// TIA Portal project "COMPACTADOR" (V21)

(* hardware
DEVICE "S7-1200 station_1"  S7-1200 Station
   slot 0: "Rack_0"  S7-1200 Rack  Rack  V1.0
   slot 1: "PLC_1"  CPU 1214C DC/DC/DC  6ES7 214-1AG40-0XB0  V4.6
   slot 2: "DI 16x24VDC_1"  SM 1221 DI16 x 24VDC  6ES7 221-1BH32-0XB0  V2.0
   slot 3: "DI 16x24VDC_2"  SM 1221 DI16 x 24VDC  6ES7 221-1BH32-0XB0  V2.0
   slot 4: "DI 16x24VDC_3"  SM 1221 DI16 x 24VDC  6ES7 221-1BH32-0XB0  V2.0
   slot 5: "DQ 16xRelay_1"  SM 1222 DQ16 x relay  6ES7 222-1HH32-0XB0  V2.0
*)

// ===== PLC "PLC_1"  CPU 1214C DC/DC/DC =====

VAR_GLOBAL   // PLC tag table "Default tag table"
   "Name" AT Logical Address : Data Type;   // Comment
END_VAR

VAR_GLOBAL   // PLC tag table "Entradas_CPU_Local"
   "STOP7" AT %I0.0 : Bool;   // Paragem Local / Botao Cogumelo de Paragem Geral (Contacto NF)
   "START" AT %I0.1 : Bool;   // Botao de Arranque do Sistema (Contacto NA)
   "AVANCA" AT %I0.2 : Bool;   // Botao Manual de Avanco do Cilindro Hidraulico (Contacto NA)
   "RECUA" AT %I0.3 : Bool;   // Botao Manual de Recuo do Cilindro Hidraulico (Contacto NA)
   "FR1" AT %I0.4 : Bool;   // Disparo / Auxiliar do Rele Termico do Motor M1 (Contacto NF)
   "FR2" AT %I0.5 : Bool;   // Disparo / Auxiliar do Rele Termico do Motor M2 (Contacto NF)
   "FR3" AT %I0.6 : Bool;   // Disparo / Auxiliar do Rele Termico do Motor M3 (Contacto NF)
   "FR4" AT %I0.7 : Bool;   // Disparo / Auxiliar do Rele Termico do Motor M4 (Contacto NF)
   "FR5" AT %I1.0 : Bool;   // Disparo / Auxiliar do Rele Termico do Motor M5 (Contacto NF)
   "FR6" AT %I1.1 : Bool;   // Disparo / Auxiliar do Rele Termico da Bomba M6 (Contacto NF)
   "SEL_AUTO" AT %I1.2 : Bool;   // Chave Seletora Auto/Manual - Posicao Automatico (Contacto NA)
   "SEL_MANUAL" AT %I1.3 : Bool;   // Chave Seletora Auto/Manual - Posicao Manual (Contacto NA)
   "RESERVA_I1_4" AT %I1.4 : Bool;   // Reserva Tecnica Local CPU
   "RESERVA_I1_5" AT %I1.5 : Bool;   // Reserva Tecnica Local CPU
END_VAR

VAR_GLOBAL   // PLC tag table "Entradas_Expansao1_SM1221"
   "SIN_Y7_COMP" AT %I2.0 : Bool;   // Diagnostico de Seguranca do Compactador (Rele IFM Y7)
   "NA_S1_COMP" AT %I2.1 : Bool;   // Interlock / Fim de Curso de Seguranca 1 do Compactador
   "NA_S2_COMP" AT %I2.2 : Bool;   // Interlock / Fim de Curso de Seguranca 2 do Compactador
   "NA_S3_COMP" AT %I2.3 : Bool;   // Interlock / Fim de Curso de Seguranca 3 do Compactador
   "SIN_Y7_M1" AT %I2.4 : Bool;   // Diagnostico de Seguranca do Motor M1 (Rele IFM Y7)
   "NA_STOP_M1" AT %I2.5 : Bool;   // Botao / Paragem Local de Seguranca do Tapete M1
   "SIN_Y7_M2" AT %I2.6 : Bool;   // Diagnostico de Seguranca do Motor M2 (Rele IFM Y7)
   "SIN_Y7_M3" AT %I2.7 : Bool;   // Diagnostico de Seguranca do Motor M3 (Rele IFM Y7)
   "NA_STOP_M2" AT %I3.0 : Bool;   // Botao / Paragem Local de Seguranca do Tapete M2
   "NA_STOP_M3" AT %I3.1 : Bool;   // Botao / Paragem Local de Seguranca do Tapete M3
   "SIN_Y7_M4" AT %I3.2 : Bool;   // Diagnostico de Seguranca do Motor M4 (Rele IFM Y7)
   "NA_STOP_M4" AT %I3.3 : Bool;   // Botao / Paragem Local de Seguranca do Tapete M4
   "SIN_Y7_M5" AT %I3.4 : Bool;   // Diagnostico de Seguranca do Motor M5 (Rele IFM Y7)
   "NA_STOP_M5" AT %I3.5 : Bool;   // Botao / Paragem Local de Seguranca do Tapete M5
   "SENSOR_75_PERCENT" AT %I3.6 : Bool;   // Sensor Optoeletronico de Nivel da Moega a 75%
   "SENSOR_100_PERCENT" AT %I3.7 : Bool;   // Sensor Optoeletronico de Nivel da Moega a 100%
END_VAR

VAR_GLOBAL   // PLC tag table "Entradas_Expansao2_SM1221"
   "M1_S4" AT %I4.0 : Bool;   // Grupo Motor M1 (Tapete 1) - Sensor S4 de Posicao / Presenca
   "M1_S5" AT %I4.1 : Bool;   // Grupo Motor M1 (Tapete 1) - Sensor S5 de Posicao / Presenca
   "M1_S6" AT %I4.2 : Bool;   // Grupo Motor M1 (Tapete 1) - Sensor S6 de Posicao / Presenca
   "M2_S7" AT %I4.3 : Bool;   // Grupo Motor M2 (Tapete 2) - Sensor S7 de Posicao / Presenca
   "M2_S8" AT %I4.4 : Bool;   // Grupo Motor M2 (Tapete 2) - Sensor S8 de Posicao / Presenca
   "M2_S9" AT %I4.5 : Bool;   // Grupo Motor M2 (Tapete 2) - Sensor S9 de Posicao / Presenca
   "M3_S10" AT %I4.6 : Bool;   // Grupo Motor M3 (Tapete 3) - Sensor S10 de Posicao / Presenca
   "M3_S11" AT %I4.7 : Bool;   // Grupo Motor M3 (Tapete 3) - Sensor S11 de Posicao / Presenca
   "M3_S12" AT %I5.0 : Bool;   // Grupo Motor M3 (Tapete 3) - Sensor S12 de Posicao / Presenca
   "M4_S13" AT %I5.1 : Bool;   // Grupo Motor M4 (Tapete 4) - Sensor S13 de Posicao / Presenca
   "M4_S14" AT %I5.2 : Bool;   // Grupo Motor M4 (Tapete 4) - Sensor S14 de Posicao / Presenca
   "M4_S15" AT %I5.3 : Bool;   // Grupo Motor M4 (Tapete 4) - Sensor S15 de Posicao / Presenca
   "M5_S16" AT %I5.4 : Bool;   // Grupo Motor M5 (Tapete 5) - Sensor S16 de Posicao / Presenca
   "M5_S17" AT %I5.5 : Bool;   // Grupo Motor M5 (Tapete 5) - Sensor S17 de Posicao / Presenca
   "M5_S18" AT %I5.6 : Bool;   // Grupo Motor M5 (Tapete 5) - Sensor S18 de Posicao / Presenca
   "M5_S19" AT %I5.7 : Bool;   // Grupo Motor M5 (Tapete 5) - Sensor S19 de Posicao / Presenca
END_VAR

VAR_GLOBAL   // PLC tag table "Entradas_Expansao3_SM1221"
   "S20_COMP" AT %I6.0 : Bool;   // Sensor de Proximidade Adicional 20 do Compactador
   "S21_COMP" AT %I6.1 : Bool;   // Sensor de Proximidade Adicional 21 do Compactador
   "STOP6_GERAL" AT %I6.2 : Bool;   // Paragem Local / Botao Cogumelo de Paragem Geral (Contacto NF)
   "RESERVA_I6_5" AT %I6.5 : Bool;   // Reserva Tecnica Modulo DI 3
   "RESERVA_I6_6" AT %I6.6 : Bool;   // Reserva Tecnica Modulo DI 3
   "RESERVA_I6_7" AT %I6.7 : Bool;   // Reserva Tecnica Modulo DI 3
   "RESERVA_I7_0" AT %I7.0 : Bool;   // Reserva Tecnica Modulo DI 3
   "RESERVA_I7_1" AT %I7.1 : Bool;   // Reserva Tecnica Modulo DI 3
   "RESERVA_I7_2" AT %I7.2 : Bool;   // Reserva Tecnica Modulo DI 3
   "RESERVA_I7_3" AT %I7.3 : Bool;   // Reserva Tecnica Modulo DI 3
   "RESERVA_I7_4" AT %I7.4 : Bool;   // Reserva Tecnica Modulo DI 3
   "RESERVA_I7_5" AT %I7.5 : Bool;   // Reserva Tecnica Modulo DI 3
   "RESERVA_I7_6" AT %I7.6 : Bool;   // Reserva Tecnica Modulo DI 3
   "RESERVA_I7_7" AT %I7.7 : Bool;   // Reserva Tecnica Modulo DI 3
   "NA_STOP_COMP" AT %I6.3 : Bool;   // Botao / Paragem Local de Seguranca do Compactador
   "RESERVA_I6_4" AT %I6.4 : Bool;   // Reserva Tecnica Modulo DI 3
END_VAR

VAR_GLOBAL   // PLC tag table "Saidas_CPU_Local"
   "KM1" AT %Q0.0 : Bool;   // Contactor de Processo do Motor M1 (Tapete 1)
   "KM2" AT %Q0.1 : Bool;   // Contactor de Processo do Motor M2 (Tapete 2)
   "KM3" AT %Q0.2 : Bool;   // Contactor de Processo do Motor M3 (Tapete 3)
   "KM4" AT %Q0.3 : Bool;   // Contactor de Processo do Motor M4 (Tapete 4)
   "KM5" AT %Q0.4 : Bool;   // Contactor de Processo do Motor M5 (Tapete 5)
   "START_SS_M6" AT %Q0.5 : Bool;   // Sinal de Habilitacao / Start da Soft Starter (Bomba M6)
   "Y1_AVANCA" AT %Q0.6 : Bool;   // Eletrovalvula de Avanco do Cilindro Hidraulico
   "Y2_RECUA" AT %Q0.7 : Bool;   // Eletrovalvula de Recuo do Cilindro Hidraulico
   "H1_VERDE" AT %Q1.0 : Bool;   // Sinalizador Luminoso Verde: Linha em Funcionamento / Automatico
   "H2_AMARELO" AT %Q1.1 : Bool;   // Sinalizador Luminoso Amarelo: Estado de Prontidao / Standby
END_VAR

VAR_GLOBAL   // PLC tag table "Saidas_Expansao1_SM1222"
   "H13_AUTO" AT %Q2.0 : Bool;   // Sinalizador: Modo AUTOMATICO Selecionado
   "H14_MANUAL" AT %Q2.1 : Bool;   // Sinalizador: Modo MANUAL Selecionado
   "H3_AZUL" AT %Q2.3 : Bool;   // Sinalizador Azul: Nivel da Moega a 75%
   "H4_VERMELHO" AT %Q2.4 : Bool;   // Sinalizador Vermelho: Nivel da Moega a 100%
   "H5_VERMELHO" AT %Q2.5 : Bool;   // Sinalizador Vermelho: Paragem / Avaria Geral da Linha
   "H6_VERMELHO" AT %Q2.6 : Bool;   // Sinalizador Vermelho: Paragem / Avaria do Compactador
   "H7_VERMELHO" AT %Q2.7 : Bool;   // Sinalizador Vermelho: Paragem / Avaria do Motor M1
   "H8_VERMELHO" AT %Q3.0 : Bool;   // Sinalizador Vermelho: Paragem / Avaria do Motor M2
   "H9_VERMELHO" AT %Q3.1 : Bool;   // Sinalizador Vermelho: Paragem / Avaria do Motor M3
   "H10_VERMELHO" AT %Q3.2 : Bool;   // Sinalizador Vermelho: Paragem / Avaria do Motor M4
   "H11_VERMELHO" AT %Q3.3 : Bool;   // Sinalizador Vermelho: Paragem / Avaria do Motor M5
   "H12_VERMELHO" AT %Q3.4 : Bool;   // Sinalizador Vermelho: Paragem / Avaria da Bomba M6
   "RESERVA_Q2_2" AT %Q2.2 : Bool;   // Reserva Tecnica Modulo DQ 1
   "RESERVA_Q3_5" AT %Q3.5 : Bool;   // Reserva Tecnica Modulo DQ 1
   "RESERVA_Q3_6" AT %Q3.6 : Bool;   // Reserva Tecnica Modulo DQ 1
   "RESERVA_Q3_7" AT %Q3.7 : Bool;   // Reserva Tecnica Modulo DQ 1
END_VAR

VAR_GLOBAL   // PLC tag table "Marcadores_Internos"
   "OK_SISTEMA" AT %M0.0 : Bool;   // Permissivo geral do sistema (calculado em FC1)
   "AUT_LINHA_LIGADA" AT %M0.1 : Bool;   // Selo da linha em modo automatico (FC3)
   "MODO_MANUAL" AT %M0.2 : Bool;   // Modo manual selecionado (FC2)
   "CICLO_RECUO" AT %M0.3 : Bool;   // Ciclo de recuo do cilindro hidraulico (FC4)
   "EMERGENCIA" AT %M0.4 : Bool;   // Paragem de emergencia ativa (FC1)
   "ETAPA_GRAFCET" AT %MW2 : Word;   // Variavel de etapa atual do GRAFCET (FC5_GRAFCET)
   "INATIVIDADE_ATIVA" AT %M0.5 : Bool;   // Timer de inatividade ativo; linha sem material durante 30 s
END_VAR

DATA_BLOCK "DB_LinhaCompactador"   // DB1
{ S7_Optimized_Access := 'TRUE' }
VERSION : 0.1
// stored: InstanceOfName FB_LinhaCompactador
"FB_LinhaCompactador"
BEGIN
END_DATA_BLOCK

FUNCTION_BLOCK "FB_LinhaCompactador"   // FB1, SCL
{ S7_Optimized_Access := 'TRUE' }
VERSION : 0.1
   VAR
      T_Start_M6 : TON_TIME;
      T_Start_M5 : TON_TIME;
      T_Start_M34 : TON_TIME;
      T_Stop_M12 : TON_TIME;
      T_Stop_M34 : TON_TIME;
      T_Stop_M5 : TON_TIME;
      T_Inatividade : TON_TIME;
   END_VAR
   VAR_TEMP
      AutoOk : Bool;
      FaultM1 : Bool;
      FaultM2 : Bool;
      FaultM3 : Bool;
      FaultM4 : Bool;
      FaultM5 : Bool;
      FaultM6 : Bool;
      FaultComp : Bool;
      EmptyM3M4 : Bool;
      EmptyM5 : Bool;
      ManualMove : Bool;
      FrontFreeM1 : Bool;
      FrontFreeM2 : Bool;
      FrontFreeM3 : Bool;
      FrontFreeM4 : Bool;
      FrontFreeM5 : Bool;
      ContentorLivre : Bool;
      LinhaSemMaterial : Bool;
   END_VAR
BEGIN

       // FC1 - Seguranca geral
       "OK_SISTEMA" :=
           "STOP7" AND
           "STOP6_GERAL" AND
           "FR1" AND
           "FR2" AND
           "FR3" AND
           "FR4" AND
           "FR5" AND
           "FR6" AND
           "SIN_Y7_COMP" AND
           "SIN_Y7_M1" AND
           "SIN_Y7_M2" AND
           "SIN_Y7_M3" AND
           "SIN_Y7_M4" AND
           "SIN_Y7_M5" AND
           "NA_STOP_M1" AND
           "NA_STOP_M2" AND
           "NA_STOP_M3" AND
           "NA_STOP_M4" AND
           "NA_STOP_M5" AND
           "NA_STOP_COMP";

       "EMERGENCIA" := NOT "OK_SISTEMA";

       // FC2 - Selecao de modo
       #AutoOk := "SEL_AUTO" AND NOT "SEL_MANUAL" AND "OK_SISTEMA";
       "MODO_MANUAL" := "SEL_MANUAL" AND NOT "SEL_AUTO" AND "OK_SISTEMA";
       "H13_AUTO" := "SEL_AUTO" AND NOT "SEL_MANUAL";
       "H14_MANUAL" := "SEL_MANUAL" AND NOT "SEL_AUTO";

       // Diagnosticos por grupo
       #FaultM1 := NOT "FR1" OR NOT "NA_STOP_M1" OR NOT "SIN_Y7_M1";
       #FaultM2 := NOT "FR2" OR NOT "NA_STOP_M2" OR NOT "SIN_Y7_M2";
       #FaultM3 := NOT "FR3" OR NOT "NA_STOP_M3" OR NOT "SIN_Y7_M3";
       #FaultM4 := NOT "FR4" OR NOT "NA_STOP_M4" OR NOT "SIN_Y7_M4";
       #FaultM5 := NOT "FR5" OR NOT "NA_STOP_M5" OR NOT "SIN_Y7_M5";
       #FaultM6 := NOT "FR6";
       #FaultComp := NOT "NA_STOP_COMP" OR NOT "SIN_Y7_COMP";

       // FC6 - Nivel da moega
       "H3_AZUL" := "SENSOR_75_PERCENT";
       "H4_VERMELHO" := "SENSOR_100_PERCENT";

       #EmptyM3M4 :=
           NOT "M3_S10" AND NOT "M3_S11" AND NOT "M3_S12" AND
           NOT "M4_S13" AND NOT "M4_S14" AND NOT "M4_S15";

       #EmptyM5 :=
           NOT "M5_S16" AND NOT "M5_S17" AND NOT "M5_S18" AND NOT "M5_S19";

       #ManualMove := "MODO_MANUAL" AND (("AVANCA" AND NOT "RECUA") OR ("RECUA" AND NOT "AVANCA"));

       // Anti-acumulacao / anti-queda: o tapete de tras so alimenta se a zona da frente estiver livre.
       #FrontFreeM1 := NOT "M3_S10" AND NOT "M3_S11" AND NOT "M3_S12";
       #FrontFreeM2 := NOT "M4_S13" AND NOT "M4_S14" AND NOT "M4_S15";
       #FrontFreeM3 := NOT "M5_S16" AND NOT "M5_S17";
       #FrontFreeM4 := NOT "M5_S18" AND NOT "M5_S19";
       #FrontFreeM5 := NOT "SENSOR_100_PERCENT";
       #ContentorLivre := NOT "S20_COMP" AND NOT "S21_COMP";
       #LinhaSemMaterial :=
           NOT "M1_S4" AND NOT "M1_S5" AND NOT "M1_S6" AND
           NOT "M2_S7" AND NOT "M2_S8" AND NOT "M2_S9" AND
           NOT "M3_S10" AND NOT "M3_S11" AND NOT "M3_S12" AND
           NOT "M4_S13" AND NOT "M4_S14" AND NOT "M4_S15" AND
           NOT "M5_S16" AND NOT "M5_S17" AND NOT "M5_S18" AND NOT "M5_S19" AND
           NOT "S20_COMP" AND NOT "S21_COMP" AND
           NOT "SENSOR_75_PERCENT" AND NOT "SENSOR_100_PERCENT";

       // Timers de arranque/paragem em cascata
       #T_Start_M6(IN := (#AutoOk AND #ContentorLivre AND ("ETAPA_GRAFCET" = WORD#16#000A)), PT := T#3s);
       #T_Start_M5(IN := (#AutoOk AND #ContentorLivre AND ("ETAPA_GRAFCET" = WORD#16#0014)), PT := T#2s);
       #T_Start_M34(IN := (#AutoOk AND #ContentorLivre AND ("ETAPA_GRAFCET" = WORD#16#001E)), PT := T#2s);
       #T_Stop_M12(IN := ("ETAPA_GRAFCET" = WORD#16#0064), PT := T#2s);
       #T_Stop_M34(IN := ("ETAPA_GRAFCET" = WORD#16#006E), PT := T#2s);
       #T_Stop_M5(IN := ("ETAPA_GRAFCET" = WORD#16#0078), PT := T#2s);
       #T_Inatividade(IN := (#AutoOk AND "AUT_LINHA_LIGADA" AND #LinhaSemMaterial), PT := T#30s);
       "INATIVIDADE_ATIVA" := #T_Inatividade.Q;

       // Prioridade maxima: emergencia ou modo invalido
       IF "EMERGENCIA" OR ("SEL_AUTO" AND "SEL_MANUAL") THEN
           "KM1" := FALSE;
           "KM2" := FALSE;
           "KM3" := FALSE;
           "KM4" := FALSE;
           "KM5" := FALSE;
           "START_SS_M6" := FALSE;
           "Y1_AVANCA" := FALSE;
           "Y2_RECUA" := FALSE;
           "AUT_LINHA_LIGADA" := FALSE;
           "CICLO_RECUO" := FALSE;
           "ETAPA_GRAFCET" := WORD#16#0000;

       ELSIF "MODO_MANUAL" THEN
           // FC4 - Manual do compactador, com intertravamento avanca/recuo
           "AUT_LINHA_LIGADA" := FALSE;
           "ETAPA_GRAFCET" := WORD#16#0000;
           "KM1" := FALSE;
           "KM2" := FALSE;
           "KM3" := FALSE;
           "KM4" := FALSE;
           "KM5" := FALSE;
           "START_SS_M6" := #ManualMove;
           "Y1_AVANCA" := "AVANCA" AND NOT "RECUA" AND "OK_SISTEMA";
           "Y2_RECUA" := "RECUA" AND NOT "AVANCA" AND "OK_SISTEMA";

       ELSIF #AutoOk THEN
           // FC3 - Automatico com arranque/paragem em cascata
           IF ("ETAPA_GRAFCET" = WORD#16#0000) AND "START" AND NOT "SENSOR_100_PERCENT" AND #ContentorLivre THEN
               "ETAPA_GRAFCET" := WORD#16#000A;
           END_IF;

           IF (("ETAPA_GRAFCET" = WORD#16#0028) AND (NOT "SEL_AUTO" OR "SENSOR_100_PERCENT" OR "INATIVIDADE_ATIVA")) THEN
               "ETAPA_GRAFCET" := WORD#16#0064;
           END_IF;

           IF ("ETAPA_GRAFCET" = WORD#16#000A) AND #T_Start_M6.Q THEN
               "ETAPA_GRAFCET" := WORD#16#0014;
           ELSIF ("ETAPA_GRAFCET" = WORD#16#0014) AND #T_Start_M5.Q THEN
               "ETAPA_GRAFCET" := WORD#16#001E;
           ELSIF ("ETAPA_GRAFCET" = WORD#16#001E) AND #T_Start_M34.Q THEN
               "ETAPA_GRAFCET" := WORD#16#0028;
               "AUT_LINHA_LIGADA" := TRUE;
           ELSIF ("ETAPA_GRAFCET" = WORD#16#0064) AND (#T_Stop_M12.Q OR #EmptyM3M4) THEN
               "ETAPA_GRAFCET" := WORD#16#006E;
           ELSIF ("ETAPA_GRAFCET" = WORD#16#006E) AND (#T_Stop_M34.Q OR #EmptyM5) THEN
               "ETAPA_GRAFCET" := WORD#16#0078;
           ELSIF ("ETAPA_GRAFCET" = WORD#16#0078) AND #T_Stop_M5.Q THEN
               "ETAPA_GRAFCET" := WORD#16#0000;
               "AUT_LINHA_LIGADA" := FALSE;
           END_IF;

           "START_SS_M6" := ("ETAPA_GRAFCET" <> WORD#16#0000) AND NOT #FaultM6 AND NOT #FaultComp;

           "KM5" :=
               (("ETAPA_GRAFCET" = WORD#16#0014) OR
                ("ETAPA_GRAFCET" = WORD#16#001E) OR
                ("ETAPA_GRAFCET" = WORD#16#0028) OR
                ("ETAPA_GRAFCET" = WORD#16#0064) OR
                ("ETAPA_GRAFCET" = WORD#16#006E)) AND
               #ContentorLivre AND
               #FrontFreeM5 AND
               NOT #FaultM5;

           "KM3" :=
               (("ETAPA_GRAFCET" = WORD#16#001E) OR
                ("ETAPA_GRAFCET" = WORD#16#0028) OR
                ("ETAPA_GRAFCET" = WORD#16#0064)) AND
               #ContentorLivre AND
               #FrontFreeM3 AND
               NOT #FaultM3 AND NOT #FaultM5;

           "KM4" :=
               (("ETAPA_GRAFCET" = WORD#16#001E) OR
                ("ETAPA_GRAFCET" = WORD#16#0028) OR
                ("ETAPA_GRAFCET" = WORD#16#0064)) AND
               #ContentorLivre AND
               #FrontFreeM4 AND
               NOT #FaultM4 AND NOT #FaultM5;

           "KM1" :=
               ("ETAPA_GRAFCET" = WORD#16#0028) AND
               #ContentorLivre AND
               NOT "SENSOR_100_PERCENT" AND
               #FrontFreeM1 AND
               NOT #FaultM1 AND NOT #FaultM3 AND NOT #FaultM5;

           "KM2" :=
               ("ETAPA_GRAFCET" = WORD#16#0028) AND
               #ContentorLivre AND
               NOT "SENSOR_100_PERCENT" AND
               #FrontFreeM2 AND
               NOT #FaultM2 AND NOT #FaultM4 AND NOT #FaultM5;

           // Ciclo basico do compactador. S20/S21 monitoram o contentor e nao sao fins de curso.
           IF "NA_S2_COMP" THEN
               "CICLO_RECUO" := TRUE;
           ELSIF "NA_S1_COMP" THEN
               "CICLO_RECUO" := FALSE;
           END_IF;

           "Y1_AVANCA" := "START_SS_M6" AND NOT "CICLO_RECUO" AND NOT "NA_S2_COMP";
           "Y2_RECUA" := "START_SS_M6" AND "CICLO_RECUO" AND NOT "NA_S1_COMP";

       ELSE
           // Sem modo valido: saidas desligadas, sistema em standby.
           "KM1" := FALSE;
           "KM2" := FALSE;
           "KM3" := FALSE;
           "KM4" := FALSE;
           "KM5" := FALSE;
           "START_SS_M6" := FALSE;
           "Y1_AVANCA" := FALSE;
           "Y2_RECUA" := FALSE;
           "AUT_LINHA_LIGADA" := FALSE;
           "ETAPA_GRAFCET" := WORD#16#0000;
       END_IF;

       // FC7 - Sinalizacao
       "H1_VERDE" := #AutoOk AND "AUT_LINHA_LIGADA" AND #ContentorLivre;
       "H2_AMARELO" := "OK_SISTEMA" AND (NOT "AUT_LINHA_LIGADA" OR NOT #ContentorLivre);
       "H6_VERMELHO" := #FaultComp;
       "H7_VERMELHO" := #FaultM1;
       "H8_VERMELHO" := #FaultM2;
       "H9_VERMELHO" := #FaultM3;
       "H10_VERMELHO" := #FaultM4;
       "H11_VERMELHO" := #FaultM5;
       "H12_VERMELHO" := #FaultM6;
       "H5_VERMELHO" :=
           "EMERGENCIA" OR
           ("SEL_AUTO" AND "SEL_MANUAL") OR
           #FaultComp OR #FaultM1 OR #FaultM2 OR #FaultM3 OR #FaultM4 OR #FaultM5 OR #FaultM6;
END_FUNCTION_BLOCK

FUNCTION "FC_LinhaCompactador_LAD" : Void   // FC21, LAD
{ S7_Optimized_Access := 'TRUE' }
VERSION : 0.1
// Visualizacao LAD da logica principal. A sequencia temporizada executavel continua em FB_LinhaCompactador.
BEGIN

REGION Network 1: FC1 - OK_SISTEMA: cadeia geral de seguranca
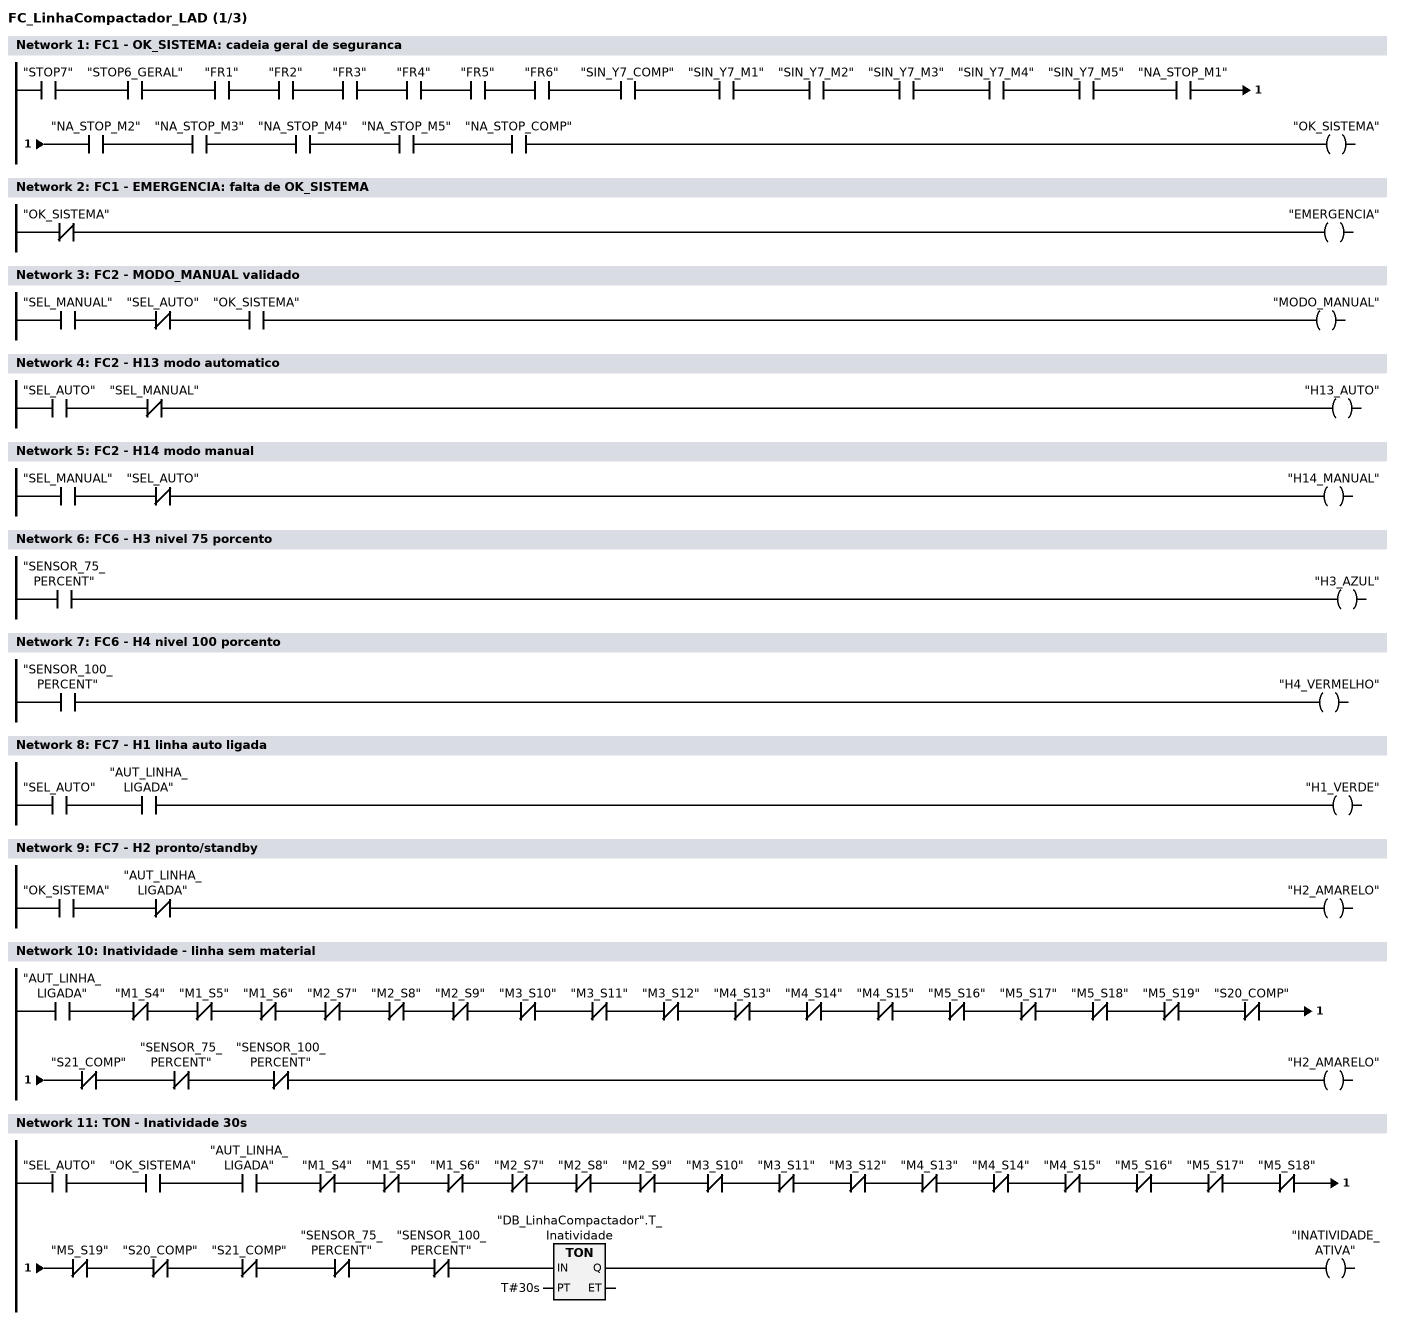
   RUNG wire#powerrail
      Contact( "STOP7" )
      Contact( "STOP6_GERAL" )
      Contact( "FR1" )
      Contact( "FR2" )
      Contact( "FR3" )
      Contact( "FR4" )
      Contact( "FR5" )
      Contact( "FR6" )
      Contact( "SIN_Y7_COMP" )
      Contact( "SIN_Y7_M1" )
      Contact( "SIN_Y7_M2" )
      Contact( "SIN_Y7_M3" )
      Contact( "SIN_Y7_M4" )
      Contact( "SIN_Y7_M5" )
      Contact( "NA_STOP_M1" )
      Contact( "NA_STOP_M2" )
      Contact( "NA_STOP_M3" )
      Contact( "NA_STOP_M4" )
      Contact( "NA_STOP_M5" )
      Contact( "NA_STOP_COMP" )
      Coil( "OK_SISTEMA" )
   END_RUNG
   // the same network as SCL:
   "OK_SISTEMA" := "STOP7" AND "STOP6_GERAL" AND "FR1" AND "FR2" AND "FR3" AND "FR4" AND "FR5" AND "FR6" AND "SIN_Y7_COMP" AND "SIN_Y7_M1" AND "SIN_Y7_M2" AND "SIN_Y7_M3" AND "SIN_Y7_M4" AND "SIN_Y7_M5" AND "NA_STOP_M1" AND "NA_STOP_M2" AND "NA_STOP_M3" AND "NA_STOP_M4" AND "NA_STOP_M5" AND "NA_STOP_COMP";
END_REGION

REGION Network 2: FC1 - EMERGENCIA: falta de OK_SISTEMA
   RUNG wire#powerrail
      I_Contact( "OK_SISTEMA" )
      Coil( "EMERGENCIA" )
   END_RUNG
   // the same network as SCL:
   "EMERGENCIA" := NOT "OK_SISTEMA";
END_REGION

REGION Network 3: FC2 - MODO_MANUAL validado
   RUNG wire#powerrail
      Contact( "SEL_MANUAL" )
      I_Contact( "SEL_AUTO" )
      Contact( "OK_SISTEMA" )
      Coil( "MODO_MANUAL" )
   END_RUNG
   // the same network as SCL:
   "MODO_MANUAL" := "SEL_MANUAL" AND NOT "SEL_AUTO" AND "OK_SISTEMA";
END_REGION

REGION Network 4: FC2 - H13 modo automatico
   RUNG wire#powerrail
      Contact( "SEL_AUTO" )
      I_Contact( "SEL_MANUAL" )
      Coil( "H13_AUTO" )
   END_RUNG
   // the same network as SCL:
   "H13_AUTO" := "SEL_AUTO" AND NOT "SEL_MANUAL";
END_REGION

REGION Network 5: FC2 - H14 modo manual
   RUNG wire#powerrail
      Contact( "SEL_MANUAL" )
      I_Contact( "SEL_AUTO" )
      Coil( "H14_MANUAL" )
   END_RUNG
   // the same network as SCL:
   "H14_MANUAL" := "SEL_MANUAL" AND NOT "SEL_AUTO";
END_REGION

REGION Network 6: FC6 - H3 nivel 75 porcento
   RUNG wire#powerrail
      Contact( "SENSOR_75_PERCENT" )
      Coil( "H3_AZUL" )
   END_RUNG
   // the same network as SCL:
   "H3_AZUL" := "SENSOR_75_PERCENT";
END_REGION

REGION Network 7: FC6 - H4 nivel 100 porcento
   RUNG wire#powerrail
      Contact( "SENSOR_100_PERCENT" )
      Coil( "H4_VERMELHO" )
   END_RUNG
   // the same network as SCL:
   "H4_VERMELHO" := "SENSOR_100_PERCENT";
END_REGION

REGION Network 8: FC7 - H1 linha auto ligada
   RUNG wire#powerrail
      Contact( "SEL_AUTO" )
      Contact( "AUT_LINHA_LIGADA" )
      Coil( "H1_VERDE" )
   END_RUNG
   // the same network as SCL:
   "H1_VERDE" := "SEL_AUTO" AND "AUT_LINHA_LIGADA";
END_REGION

REGION Network 9: FC7 - H2 pronto/standby
   RUNG wire#powerrail
      Contact( "OK_SISTEMA" )
      I_Contact( "AUT_LINHA_LIGADA" )
      Coil( "H2_AMARELO" )
   END_RUNG
   // the same network as SCL:
   "H2_AMARELO" := "OK_SISTEMA" AND NOT "AUT_LINHA_LIGADA";
END_REGION

REGION Network 10: Inatividade - linha sem material
   RUNG wire#powerrail
      Contact( "AUT_LINHA_LIGADA" )
      I_Contact( "M1_S4" )
      I_Contact( "M1_S5" )
      I_Contact( "M1_S6" )
      I_Contact( "M2_S7" )
      I_Contact( "M2_S8" )
      I_Contact( "M2_S9" )
      I_Contact( "M3_S10" )
      I_Contact( "M3_S11" )
      I_Contact( "M3_S12" )
      I_Contact( "M4_S13" )
      I_Contact( "M4_S14" )
      I_Contact( "M4_S15" )
      I_Contact( "M5_S16" )
      I_Contact( "M5_S17" )
      I_Contact( "M5_S18" )
      I_Contact( "M5_S19" )
      I_Contact( "S20_COMP" )
      I_Contact( "S21_COMP" )
      I_Contact( "SENSOR_75_PERCENT" )
      I_Contact( "SENSOR_100_PERCENT" )
      Coil( "H2_AMARELO" )
   END_RUNG
   // the same network as SCL:
   "H2_AMARELO" := "AUT_LINHA_LIGADA" AND NOT "M1_S4" AND NOT "M1_S5" AND NOT "M1_S6" AND NOT "M2_S7" AND NOT "M2_S8" AND NOT "M2_S9" AND NOT "M3_S10" AND NOT "M3_S11" AND NOT "M3_S12" AND NOT "M4_S13" AND NOT "M4_S14" AND NOT "M4_S15" AND NOT "M5_S16" AND NOT "M5_S17" AND NOT "M5_S18" AND NOT "M5_S19" AND NOT "S20_COMP" AND NOT "S21_COMP" AND NOT "SENSOR_75_PERCENT" AND NOT "SENSOR_100_PERCENT";
END_REGION

REGION Network 11: TON - Inatividade 30s
   "DB_LinhaCompactador".T_Inatividade.TON(IN := "SEL_AUTO" AND "OK_SISTEMA" AND "AUT_LINHA_LIGADA" AND NOT "M1_S4" AND NOT "M1_S5" AND NOT "M1_S6" AND NOT "M2_S7" AND NOT "M2_S8" AND NOT "M2_S9" AND NOT "M3_S10" AND NOT "M3_S11" AND NOT "M3_S12" AND NOT "M4_S13" AND NOT "M4_S14" AND NOT "M4_S15" AND NOT "M5_S16" AND NOT "M5_S17" AND NOT "M5_S18" AND NOT "M5_S19" AND NOT "S20_COMP" AND NOT "S21_COMP" AND NOT "SENSOR_75_PERCENT" AND NOT "SENSOR_100_PERCENT",
                           PT := T#30s);
   "INATIVIDADE_ATIVA" := "DB_LinhaCompactador".T_Inatividade.Q;
END_REGION

REGION Network 12: Manual - avanco cilindro
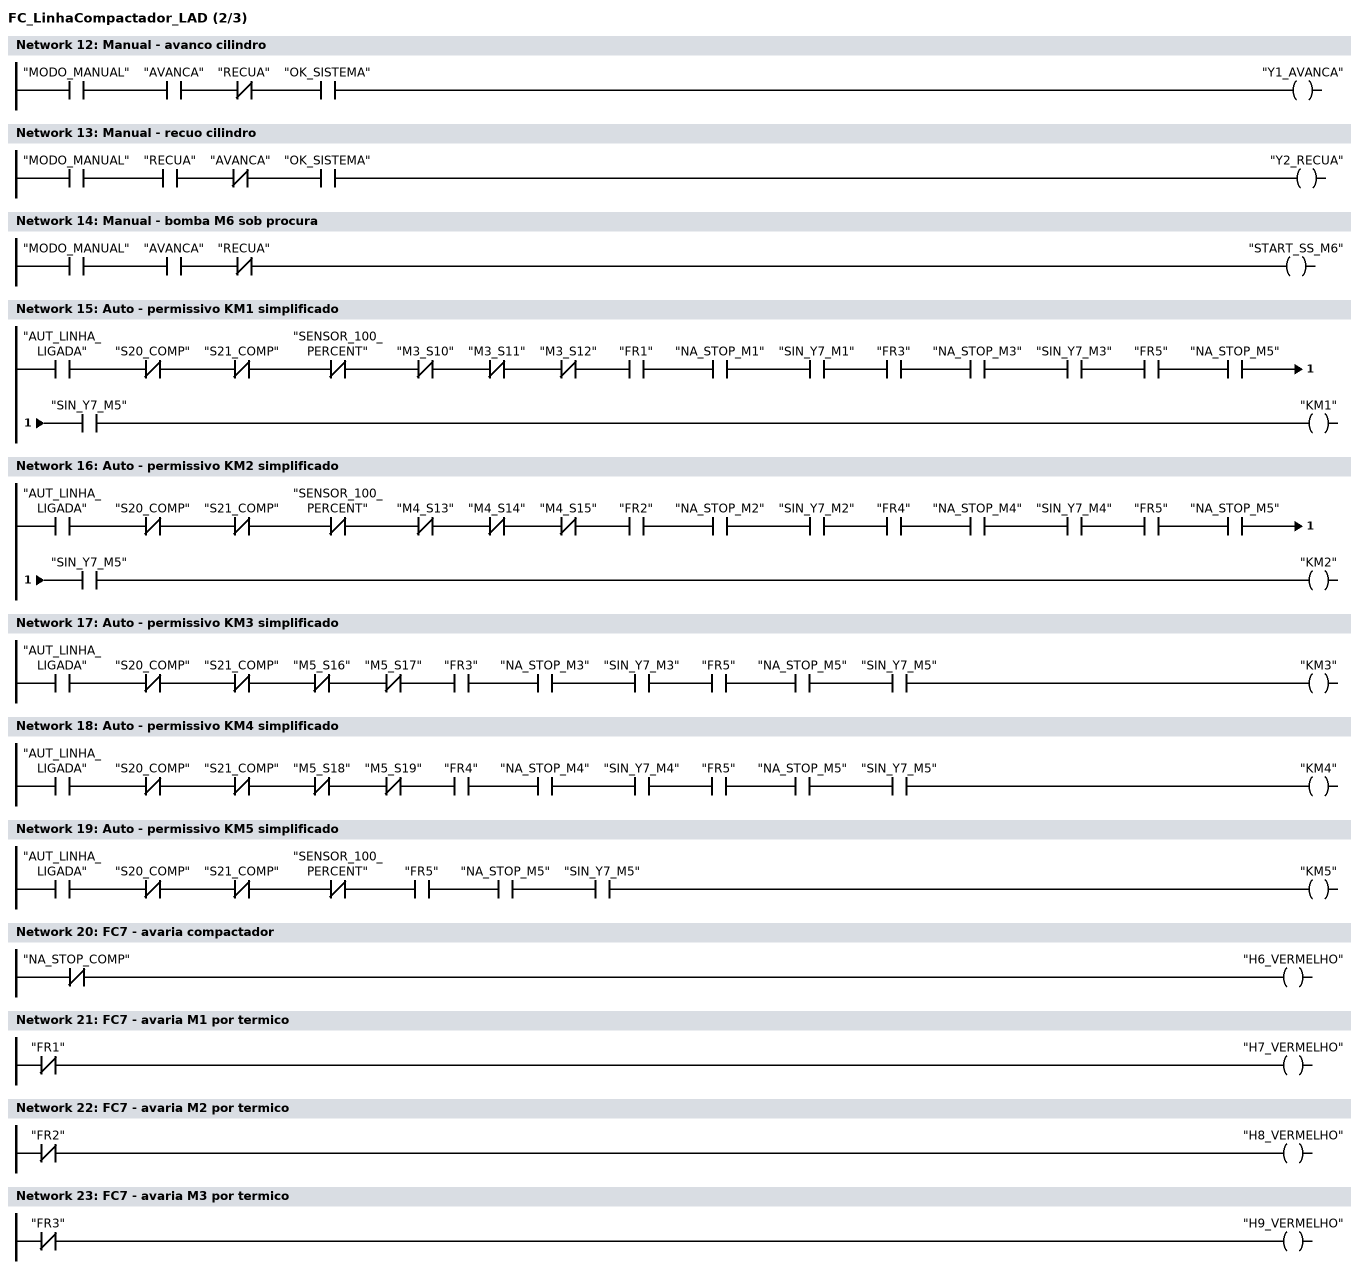
   RUNG wire#powerrail
      Contact( "MODO_MANUAL" )
      Contact( "AVANCA" )
      I_Contact( "RECUA" )
      Contact( "OK_SISTEMA" )
      Coil( "Y1_AVANCA" )
   END_RUNG
   // the same network as SCL:
   "Y1_AVANCA" := "MODO_MANUAL" AND "AVANCA" AND NOT "RECUA" AND "OK_SISTEMA";
END_REGION

REGION Network 13: Manual - recuo cilindro
   RUNG wire#powerrail
      Contact( "MODO_MANUAL" )
      Contact( "RECUA" )
      I_Contact( "AVANCA" )
      Contact( "OK_SISTEMA" )
      Coil( "Y2_RECUA" )
   END_RUNG
   // the same network as SCL:
   "Y2_RECUA" := "MODO_MANUAL" AND "RECUA" AND NOT "AVANCA" AND "OK_SISTEMA";
END_REGION

REGION Network 14: Manual - bomba M6 sob procura
   RUNG wire#powerrail
      Contact( "MODO_MANUAL" )
      Contact( "AVANCA" )
      I_Contact( "RECUA" )
      Coil( "START_SS_M6" )
   END_RUNG
   // the same network as SCL:
   "START_SS_M6" := "MODO_MANUAL" AND "AVANCA" AND NOT "RECUA";
END_REGION

REGION Network 15: Auto - permissivo KM1 simplificado
   RUNG wire#powerrail
      Contact( "AUT_LINHA_LIGADA" )
      I_Contact( "S20_COMP" )
      I_Contact( "S21_COMP" )
      I_Contact( "SENSOR_100_PERCENT" )
      I_Contact( "M3_S10" )
      I_Contact( "M3_S11" )
      I_Contact( "M3_S12" )
      Contact( "FR1" )
      Contact( "NA_STOP_M1" )
      Contact( "SIN_Y7_M1" )
      Contact( "FR3" )
      Contact( "NA_STOP_M3" )
      Contact( "SIN_Y7_M3" )
      Contact( "FR5" )
      Contact( "NA_STOP_M5" )
      Contact( "SIN_Y7_M5" )
      Coil( "KM1" )
   END_RUNG
   // the same network as SCL:
   "KM1" := "AUT_LINHA_LIGADA" AND NOT "S20_COMP" AND NOT "S21_COMP" AND NOT "SENSOR_100_PERCENT" AND NOT "M3_S10" AND NOT "M3_S11" AND NOT "M3_S12" AND "FR1" AND "NA_STOP_M1" AND "SIN_Y7_M1" AND "FR3" AND "NA_STOP_M3" AND "SIN_Y7_M3" AND "FR5" AND "NA_STOP_M5" AND "SIN_Y7_M5";
END_REGION

REGION Network 16: Auto - permissivo KM2 simplificado
   RUNG wire#powerrail
      Contact( "AUT_LINHA_LIGADA" )
      I_Contact( "S20_COMP" )
      I_Contact( "S21_COMP" )
      I_Contact( "SENSOR_100_PERCENT" )
      I_Contact( "M4_S13" )
      I_Contact( "M4_S14" )
      I_Contact( "M4_S15" )
      Contact( "FR2" )
      Contact( "NA_STOP_M2" )
      Contact( "SIN_Y7_M2" )
      Contact( "FR4" )
      Contact( "NA_STOP_M4" )
      Contact( "SIN_Y7_M4" )
      Contact( "FR5" )
      Contact( "NA_STOP_M5" )
      Contact( "SIN_Y7_M5" )
      Coil( "KM2" )
   END_RUNG
   // the same network as SCL:
   "KM2" := "AUT_LINHA_LIGADA" AND NOT "S20_COMP" AND NOT "S21_COMP" AND NOT "SENSOR_100_PERCENT" AND NOT "M4_S13" AND NOT "M4_S14" AND NOT "M4_S15" AND "FR2" AND "NA_STOP_M2" AND "SIN_Y7_M2" AND "FR4" AND "NA_STOP_M4" AND "SIN_Y7_M4" AND "FR5" AND "NA_STOP_M5" AND "SIN_Y7_M5";
END_REGION

REGION Network 17: Auto - permissivo KM3 simplificado
   RUNG wire#powerrail
      Contact( "AUT_LINHA_LIGADA" )
      I_Contact( "S20_COMP" )
      I_Contact( "S21_COMP" )
      I_Contact( "M5_S16" )
      I_Contact( "M5_S17" )
      Contact( "FR3" )
      Contact( "NA_STOP_M3" )
      Contact( "SIN_Y7_M3" )
      Contact( "FR5" )
      Contact( "NA_STOP_M5" )
      Contact( "SIN_Y7_M5" )
      Coil( "KM3" )
   END_RUNG
   // the same network as SCL:
   "KM3" := "AUT_LINHA_LIGADA" AND NOT "S20_COMP" AND NOT "S21_COMP" AND NOT "M5_S16" AND NOT "M5_S17" AND "FR3" AND "NA_STOP_M3" AND "SIN_Y7_M3" AND "FR5" AND "NA_STOP_M5" AND "SIN_Y7_M5";
END_REGION

REGION Network 18: Auto - permissivo KM4 simplificado
   RUNG wire#powerrail
      Contact( "AUT_LINHA_LIGADA" )
      I_Contact( "S20_COMP" )
      I_Contact( "S21_COMP" )
      I_Contact( "M5_S18" )
      I_Contact( "M5_S19" )
      Contact( "FR4" )
      Contact( "NA_STOP_M4" )
      Contact( "SIN_Y7_M4" )
      Contact( "FR5" )
      Contact( "NA_STOP_M5" )
      Contact( "SIN_Y7_M5" )
      Coil( "KM4" )
   END_RUNG
   // the same network as SCL:
   "KM4" := "AUT_LINHA_LIGADA" AND NOT "S20_COMP" AND NOT "S21_COMP" AND NOT "M5_S18" AND NOT "M5_S19" AND "FR4" AND "NA_STOP_M4" AND "SIN_Y7_M4" AND "FR5" AND "NA_STOP_M5" AND "SIN_Y7_M5";
END_REGION

REGION Network 19: Auto - permissivo KM5 simplificado
   RUNG wire#powerrail
      Contact( "AUT_LINHA_LIGADA" )
      I_Contact( "S20_COMP" )
      I_Contact( "S21_COMP" )
      I_Contact( "SENSOR_100_PERCENT" )
      Contact( "FR5" )
      Contact( "NA_STOP_M5" )
      Contact( "SIN_Y7_M5" )
      Coil( "KM5" )
   END_RUNG
   // the same network as SCL:
   "KM5" := "AUT_LINHA_LIGADA" AND NOT "S20_COMP" AND NOT "S21_COMP" AND NOT "SENSOR_100_PERCENT" AND "FR5" AND "NA_STOP_M5" AND "SIN_Y7_M5";
END_REGION

REGION Network 20: FC7 - avaria compactador
   RUNG wire#powerrail
      I_Contact( "NA_STOP_COMP" )
      Coil( "H6_VERMELHO" )
   END_RUNG
   // the same network as SCL:
   "H6_VERMELHO" := NOT "NA_STOP_COMP";
END_REGION

REGION Network 21: FC7 - avaria M1 por termico
   RUNG wire#powerrail
      I_Contact( "FR1" )
      Coil( "H7_VERMELHO" )
   END_RUNG
   // the same network as SCL:
   "H7_VERMELHO" := NOT "FR1";
END_REGION

REGION Network 22: FC7 - avaria M2 por termico
   RUNG wire#powerrail
      I_Contact( "FR2" )
      Coil( "H8_VERMELHO" )
   END_RUNG
   // the same network as SCL:
   "H8_VERMELHO" := NOT "FR2";
END_REGION

REGION Network 23: FC7 - avaria M3 por termico
   RUNG wire#powerrail
      I_Contact( "FR3" )
      Coil( "H9_VERMELHO" )
   END_RUNG
   // the same network as SCL:
   "H9_VERMELHO" := NOT "FR3";
END_REGION

REGION Network 24: FC7 - avaria M4 por termico
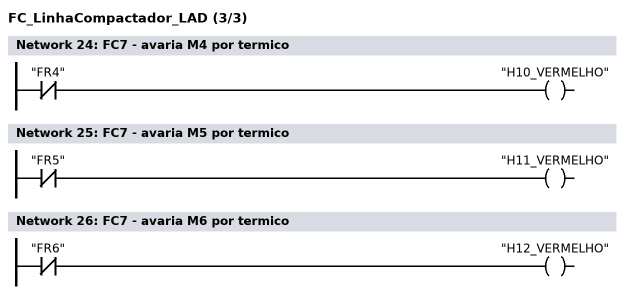
   RUNG wire#powerrail
      I_Contact( "FR4" )
      Coil( "H10_VERMELHO" )
   END_RUNG
   // the same network as SCL:
   "H10_VERMELHO" := NOT "FR4";
END_REGION

REGION Network 25: FC7 - avaria M5 por termico
   RUNG wire#powerrail
      I_Contact( "FR5" )
      Coil( "H11_VERMELHO" )
   END_RUNG
   // the same network as SCL:
   "H11_VERMELHO" := NOT "FR5";
END_REGION

REGION Network 26: FC7 - avaria M6 por termico
   RUNG wire#powerrail
      I_Contact( "FR6" )
      Coil( "H12_VERMELHO" )
   END_RUNG
   // the same network as SCL:
   "H12_VERMELHO" := NOT "FR6";
END_REGION
END_FUNCTION

ORGANIZATION_BLOCK "Main"   // OB1, SCL, ProgramCycle
TITLE = "Main Program Sweep (Cycle)"
{ S7_Optimized_Access := 'TRUE' }
VERSION : 0.1
   VAR_INPUT
      Initial_Call : Bool;   // Initial call of this OB
      Remanence : Bool;   // =True, if remanent data are available
   END_VAR
BEGIN

       "DB_LinhaCompactador"();
END_ORGANIZATION_BLOCK